FUNCTION_BLOCK INIT (* E_TRIG Counterpart *)
  (* Standard: 61131-3; Classification: standard boolean function; Description: Copyright (c) 2011 TU Wien ACIN, HR Agrartechnik GmbH This program and the accompanying materials are made available under the terms of the Eclipse Public License 2.0 which is available at https://www.eclipse.org/legal/epl-2.0/ SPDX-License-Identifier: EPL-2.0 *)
  (* Version 1.0, 2011-06-21, Monika Wenger, TU Wien ACIN, initial API and implementation and/or initial documentation *)
  (* Version 3.0, 2025-04-14, Patrick Aigner, changed package *)
  PACKAGE iec61131::booleanOperators;
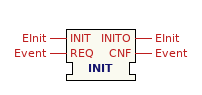
  EVENT_INPUT
    INIT : EInit; (* Initialization Request *)
    REQ; (* Service Request *)
  END_EVENT
  EVENT_OUTPUT
    INITO : EInit; (* Initialization Confirm *)
    CNF; (* Confirmation of Requested Service *)
  END_EVENT
  EVENT_CONNECTIONS
    INIT TO INITO;
    REQ TO CNF;
  END_CONNECTIONS
END_FUNCTION_BLOCK
